TYPE DUT_PPM :
STRUCT
	{attribute 'pytmc' := '
		pv: SPM
	'}
	stPowerMeter: DUT_PPM_PowerMeter;
	
	{attribute 'pytmc' := '
		pv: YAG:STC
		io: input
	'}
	fYagThermoCouple AT %I*: INT;

	{attribute 'pytmc' := '
		pv: GIGE
	'}
	stGige: DUT_PPM_Gige;

	{attribute 'pytmc' := '
		pv: CFM
	'}
	stFlowMeter: DUT_L2SI_Flowmeter;
END_STRUCT
END_TYPE

(* stored: Version 1.1.0.1, ProductVersion 3.1.4022.12
   DUT DUT_PPM: Id {f06f8092-7b61-4b55-b289-c90599f01c00} *)
